Staubli VAL3: stop.pgx

program stop()
begin
  cls()
  gotoxy(10,5)
  put("欢迎再次使用!")

end
